// TIA Portal V19 export
FUNCTION_BLOCK "CutLength"   // FB34, LAD
// stored: MemoryReserve 100, SetENOAutomatically false
   VAR_INPUT
      AreaInterface : "AreaInterface";
      CutDone : Bool;
      CutAtRest : Bool;
      MaterialCounter { ExternalAccessible := 'False'; ExternalVisible := 'False'; ExternalWritable := 'False'} : Struct
         AlrPresence : Bool;
         WngPresence : Bool;
         Data : "MatCountData";
      END_STRUCT;
   END_VAR
   VAR_OUTPUT
      CutData { ExternalAccessible := 'False'; ExternalVisible := 'False'; ExternalWritable := 'False'} : Struct
         Gap : LReal;
         MaterialPosition : LReal;
         MaterialTargetPosition : LReal;
         DeltaTarget : LReal;
         MaterialMissingToTarget : LReal;
      END_STRUCT;
   END_VAR
   VAR_IN_OUT
      TO_Carriage_MeasInput : TO_MeasuringInput;
      TO_Wheel_MeasInput : TO_MeasuringInput;
      Pers : Struct
         CarriageMeasID : UInt;
         WheelMeasID : UInt;
         CarriageEncoder : LReal;
         WheelEncoder : LReal;
         LastCut_Material_Position : LReal;
         PrevCut_Material_Position : LReal;
      END_STRUCT;
   END_VAR
   VAR
      Sts : Struct
         Status : Int;
         CarriageMeasInp_LastID : UInt;
         WheelMeasInp_LastID : UInt;
         AtCut : Struct
            Lead_Position : LReal;
            Carriage_Position : LReal;
         END_STRUCT;
      END_STRUCT;
      Alarm : Struct
         Carriage_MeasInput : "TMeasuring_Alarms";
         Wheel_MeasInput : "TMeasuring_Alarms";
         MeasInpNotEngaged { S7_SetPoint := 'True'} : Bool;
      END_STRUCT;
      Diag : Struct
         Carriage_MeasInput : "TO_Diagnostic";
         Wheel_MeasInput : "TO_Diagnostic";
      END_STRUCT;
      Carriage_MeasInp { ExternalAccessible := 'False'; ExternalVisible := 'False'; ExternalWritable := 'False'} : "MeasuringInput";
      Wheel_MeasInp { ExternalAccessible := 'False'; ExternalVisible := 'False'; ExternalWritable := 'False'} : "MeasuringInput";
      AuxPE : Struct
         CutDone : Bool;
      END_STRUCT;
      PE { ExternalAccessible := 'False'; ExternalVisible := 'False'; ExternalWritable := 'False'} : Struct
         CutDone : Bool;
      END_STRUCT;
   END_VAR
   VAR_TEMP   // added for the SCL form of the ladder/FBD networks
      _w1 : Bool;
   END_VAR
BEGIN

REGION Network 2 (SCL): Reset alarms

   IF #AreaInterface.RstAlarms THEN

       #Alarm.MeasInpNotEngaged := FALSE;

   END_IF;
END_REGION

REGION Network 3: PE Cut Done
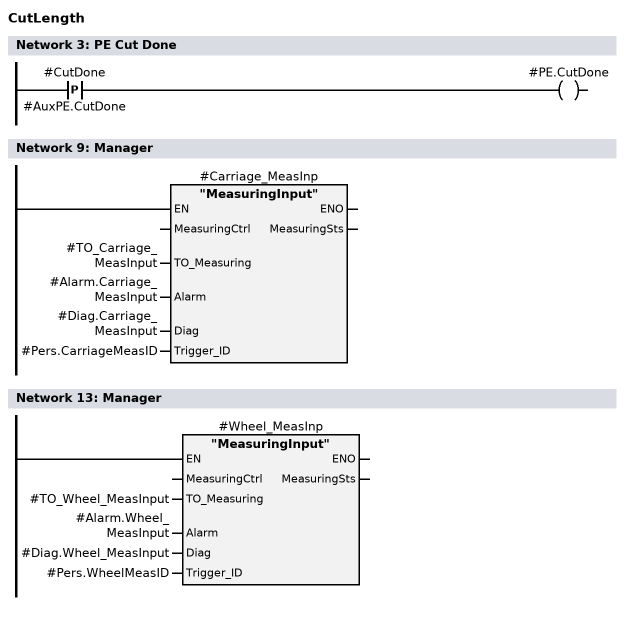
   RUNG wire#powerrail
      P_Contact(operand := #CutDone, bit := #AuxPE.CutDone)
      Coil( #PE.CutDone )
   END_RUNG
   // the same network as SCL:
   #_w1 := #CutDone AND NOT #AuxPE.CutDone;   // rising edge of #CutDone
   #AuxPE.CutDone := #CutDone;
   #PE.CutDone := #_w1;
END_REGION

REGION Network 4 (SCL)


   CASE #Sts.Status OF

       0:
           IF #CutAtRest THEN
               #Sts.CarriageMeasInp_LastID := #Pers.CarriageMeasID;
               #Sts.WheelMeasInp_LastID := #Pers.WheelMeasID;
           END_IF;

           IF #PE.CutDone THEN

               #Sts.Status += 1;
           END_IF;

       1:

           IF #Sts.CarriageMeasInp_LastID <> #Pers.CarriageMeasID AND
               #Sts.WheelMeasInp_LastID <> #Pers.WheelMeasID
           THEN

               #Pers.CarriageEncoder := #Carriage_MeasInp.MeasuringSts.MeasuringValue1;
               #Pers.WheelEncoder := #Wheel_MeasInp.MeasuringSts.MeasuringValue1;

               #Pers.PrevCut_Material_Position := #Pers.LastCut_Material_Position;

               #Sts.AtCut.Lead_Position := "PosAxisToPosMat_Wheel"(PosAxis := #Pers.WheelEncoder , Data := #MaterialCounter.Data);
               #Sts.AtCut.Carriage_Position := #Pers.CarriageEncoder;
               #Pers.LastCut_Material_Position := "M_PosAMinusCostB"(PosA := #Sts.AtCut.Lead_Position, CostB := #Sts.AtCut.Carriage_Position, MODULE := #MaterialCounter.Data.COUNTER_MODULE);

               #CutData.MaterialTargetPosition := "RollformingMng".FlyingCutoff.CIn.Target.MaterialPosition;
               #CutData.DeltaTarget := #CutData.MaterialTargetPosition - #Pers.LastCut_Material_Position;

               #CutData.MaterialMissingToTarget := "RollformingMng".FlyingCutoff.Sts.MaterialMissingToTarget;

               #Sts.Status := 0;

           ELSIF #CutAtRest THEN

               #Alarm.MeasInpNotEngaged := TRUE;
               #Sts.Status := 0;

           END_IF;

   END_CASE;


   #CutData.MaterialPosition := #Pers.LastCut_Material_Position;
   #CutData.Gap := "M_PosAMinusPosB"(PosA := #Pers.LastCut_Material_Position, PosB :=  #Pers.PrevCut_Material_Position, MODULE := #MaterialCounter.Data.COUNTER_MODULE);
END_REGION

REGION Network 7: <<< CARRIAGE MEAS INPUT >>>
END_REGION

REGION Network 8 (SCL): Control
   #Carriage_MeasInp.MeasuringCtrl.Rst := #AreaInterface.RstAlarms;
   #Carriage_MeasInp.MeasuringCtrl.MeasureEnable := NOT #AreaInterface.EStop;
   #Carriage_MeasInp.MeasuringCtrl.Mode := 0;
END_REGION

REGION Network 9: Manager
   RUNG wire#powerrail
      #Carriage_MeasInp(MeasuringCtrl :=, TO_Measuring := #TO_Carriage_MeasInput, Alarm := #Alarm.Carriage_MeasInput, Diag := #Diag.Carriage_MeasInput, Trigger_ID := #Pers.CarriageMeasID, MeasuringSts =>)
   END_RUNG
   // the same network as SCL:
   #Carriage_MeasInp(TO_Measuring := #TO_Carriage_MeasInput,   // "MeasuringInput"
                     Alarm := #Alarm.Carriage_MeasInput,
                     Diag := #Diag.Carriage_MeasInput,
                     Trigger_ID := #Pers.CarriageMeasID);
END_REGION

REGION Network 10: >
END_REGION

REGION Network 11: <<< WHEEL MEAS INPUT >>>
END_REGION

REGION Network 12 (SCL): Control
   #Wheel_MeasInp.MeasuringCtrl.Rst := #AreaInterface.RstAlarms;
   #Wheel_MeasInp.MeasuringCtrl.MeasureEnable := NOT #AreaInterface.EStop;
   #Wheel_MeasInp.MeasuringCtrl.Mode := 0;
END_REGION

REGION Network 13: Manager
   RUNG wire#powerrail
      #Wheel_MeasInp(MeasuringCtrl :=, TO_Measuring := #TO_Wheel_MeasInput, Alarm := #Alarm.Wheel_MeasInput, Diag := #Diag.Wheel_MeasInput, Trigger_ID := #Pers.WheelMeasID, MeasuringSts =>)
   END_RUNG
   // the same network as SCL:
   #Wheel_MeasInp(TO_Measuring := #TO_Wheel_MeasInput,   // "MeasuringInput"
                  Alarm := #Alarm.Wheel_MeasInput,
                  Diag := #Diag.Wheel_MeasInput,
                  Trigger_ID := #Pers.WheelMeasID);
END_REGION
END_FUNCTION_BLOCK
